{attribute 'linkalways'} 
{attribute 'no_explicit_call' := 'This FB is a CLASS and must be accessed using methods or properties'}
{attribute 'enable_dynamic_creation'}
FUNCTION_BLOCK _Array0to1OfUINT EXTENDS ArrayDatatypeBase_1D
VAR CONSTANT
	lBound : DINT := 0;
	uBound : DINT := 1;
END_VAR
VAR
	localData : ARRAY [lBound..uBound] OF UINT;
	activeData : REFERENCE TO ARRAY [lBound..uBound] OF UINT REF= localData;
	elements : ARRAY [lBound..uBound] OF _UINT(0);
	baseType : _UINT(0);
END_VAR

PROPERTY PUBLIC Address : PVOID
GET
Address := ADR(activeData);
END_GET
END_PROPERTY

PROPERTY PUBLIC BaseDatatype : I_Datatype
GET
BaseDatatype := baseType;
END_GET
END_PROPERTY

METHOD PUBLIC ClearReference
VAR_INPUT
END_VAR
activeData REF= localData;
SetElementReference();
END_METHOD

METHOD PUBLIC Clone : I_Datatype
VAR
    pClone : POINTER TO _Array0to1OfUINT;
END_VAR
pClone := __NEW(_Array0to1OfUINT());
pClone^.Value := Value;
Clone := pClone^;
END_METHOD

METHOD FB_init : BOOL
VAR_INPUT
	bInitRetains : BOOL; // if TRUE, the retain variables are initialized (warm start / cold start)
	bInCopyCode : BOOL;  // if TRUE, the instance afterwards gets moved into the copy code (online change)
END_VAR
SetElementReference();
END_METHOD

METHOD PUBLIC MakeReferenceTo
VAR_INPUT
	ReferenceTarget : REFERENCE TO ARRAY [lBound..uBound] OF UINT;
END_VAR
activeData REF= ReferenceTarget;
SetElementReference();
END_METHOD

METHOD PROTECTED OnSerializeArrayValues
VAR_INPUT
	Serializer : I_Serializer;
END_VAR
VAR
	i : DINT;
END_VAR
FOR i := lBound TO uBound DO
	elements[i].SerializeWith(Serializer);
END_FOR
END_METHOD

METHOD PROTECTED SetElementReference
VAR_INPUT
END_VAR
VAR
	i : DINT;
END_VAR
FOR i := lBound TO uBound DO
	elements[i].MakeReferenceTo(activeData[i]);
END_FOR
END_METHOD

PROPERTY PUBLIC Size : UDINT
GET
Size := SIZEOF(activeData);
END_GET
END_PROPERTY

METHOD PROTECTED TryDeserializeArrayValues : BOOL
VAR_INPUT
	Deserializer : I_Deserializer;
	Feedback : I_DeserializerFeedback;
END_VAR
VAR
	enumerator : I_DeserializerArrayForwardEnumerator;
	i : DINT;
END_VAR
enumerator := Deserializer.GetArrayEnumerator();
i := lBound;

WHILE enumerator.MoveNext() AND i <= uBound DO
	
	IF NOT elements[i].TryDeserializeFrom(enumerator.Current, Feedback) THEN
		EXIT;
	END_IF
	i := i + 1;

END_WHILE
enumerator.Dispose();
END_METHOD

METHOD PUBLIC TryGetElementAsDatatypeByIndex : BOOL
VAR_INPUT
	Index : DINT;
	Destination : REFERENCE TO I_Datatype;
END_VAR
IF Index < lbound OR Index > ubound THEN
	RETURN;
END_IF

Destination := elements[Index];
TryGetElementAsDatatypeByIndex := TRUE;
END_METHOD

METHOD PUBLIC TryGetLowerBound : BOOL
VAR_INPUT
	Dimention : UDINT;
	Destination : REFERENCE TO DINT;
END_VAR
IF Dimention = 1 THEN
	Destination := lBound;
	TryGetLowerBound := TRUE;
END_IF
END_METHOD

METHOD PUBLIC TryGetUpperBound : BOOL
VAR_INPUT
	Dimention : UDINT;
	Destination : REFERENCE TO DINT;
END_VAR
IF Dimention = 1 THEN
	Destination := uBound;
	TryGetUpperBound := TRUE;
END_IF
END_METHOD

METHOD TryMakeReferenceTo : BOOL
VAR_INPUT
	Target : I_Datatype;
END_VAR
VAR
	targetAsArray : I_ArrayDatatype;
	pTargetData : POINTER TO ARRAY [lBound..uBound] OF UINT;
END_VAR
IF NOT Target.TryResolveAsArrayDatatype(targetAsArray) THEN
	RETURN;
END_IF

IF NOT (targetAsArray.Identifier = Identifier) THEN
	RETURN;
END_IF

pTargetData := Target.Address;
activeData REF= pTargetData^;
SetElementReference();
TryMakeReferenceTo := TRUE;
END_METHOD

PROPERTY PUBLIC Value : REFERENCE TO ARRAY [lBound..uBound] OF UINT;
GET
Value ref= activeData;
END_GET
END_PROPERTY

END_FUNCTION_BLOCK

(* stored: Version 1.1.0.1, ProductVersion 3.1.4024.13
   POU _Array0to1OfUINT: Id {91f56a84-a3ad-02fb-247a-7fd72a195245}, SpecialFunc None
   Folder Core: Id {cd16623f-2f44-04f8-12ed-402eb52d23ce}
   Folder Constructor: Id {53b5f4d7-0929-07ad-0c95-dcbdd938d303}
   Folder Protected: Id {bfcd0752-dca1-010d-2654-8e80fa988d5c}
   Folder Customize: Id {93f4853e-3291-0209-3b0d-3a03217bffec}
   Property Address: Id {e4be0ecd-1da8-09a7-3ba4-462a96011d6f}
   Get Get: Id {10ac5d7b-97a8-0acb-1ed0-f8e435d7c940}
   Property BaseDatatype: Id {edb00700-2f2e-0319-1cfa-fda738933037}
   Get Get: Id {9722c95f-91af-0dcb-3fe4-37c19b6854d1}
   Method ClearReference: Id {db457f0a-8653-0eb9-0bf9-33540f165d24}
   Method Clone: Id {34284eb2-0911-0fb5-3b12-ddc89fd98657}
   Method FB_init: Id {b3f2ba8b-1aeb-0446-22c4-c8e821b28b3d}
   Method MakeReferenceTo: Id {50979fb1-417b-0364-29ea-a7b1be9f1864}
   Method OnSerializeArrayValues: Id {d6a1210b-bd6d-0a1b-10d9-aa22947ce627}
   Method SetElementReference: Id {63ac74b9-e2cd-0d80-14a4-3301fa9df654}
   Property Size: Id {492f15c5-e2a6-0c20-3a53-d2e7f7016092}
   Get Get: Id {6250446f-5a22-0ab7-3c45-c5a58d8bf85b}
   Method TryDeserializeArrayValues: Id {3d510fe8-3456-0b3a-3be8-22856ce57d7b}
   Method TryGetElementAsDatatypeByIndex: Id {5a0949a3-3ef8-031d-2529-5692a84fd58b}
   Method TryGetLowerBound: Id {968d7999-983a-03f3-275d-df5e50d5eac5}
   Method TryGetUpperBound: Id {e2db770a-42a9-03b6-1f07-e6458571e3ec}
   Method TryMakeReferenceTo: Id {53baf4de-986b-0f6c-1f49-f67f967481c1}
   Property Value: Id {f6274510-629d-0df8-271a-06095cda6daf}
   Get Get: Id {ddfadefc-caf4-04f4-1a47-677d8eaec957} *)
